FUNCTION_BLOCK VariableToEvent (* Basic Function Block Type *)
  (* Standard: 61499-2 *)
  (* Version 0.2, 2003-12-04, JHC, Rockwell Automation, Renamed for better indexing. *)
  (* Version 0.1, 2002-11-05, JHC, Rockwell Automation, Corrected missing ST element in Algorithm REQ. *)
  (* Version 0.0, 2000-05-30, JHC, Rockwell Automation *)
  (* Compiler header: package fb.rt.cs725; *)
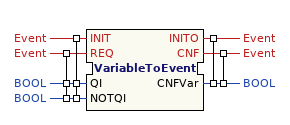
  EVENT_INPUT
    INIT WITH QI, NOTQI; (* Initialization Request *)
    REQ WITH QI, NOTQI; (* Normal Execution Request *)
  END_EVENT
  EVENT_OUTPUT
    INITO WITH CNFVar; (* Initialization Confirm *)
    CNF WITH CNFVar; (* Execution Confirmation *)
  END_EVENT
  VAR_INPUT
    QI : BOOL; (* Input event qualifier *)
    NOTQI : BOOL;
  END_VAR
  VAR_OUTPUT
    CNFVar : BOOL;
  END_VAR
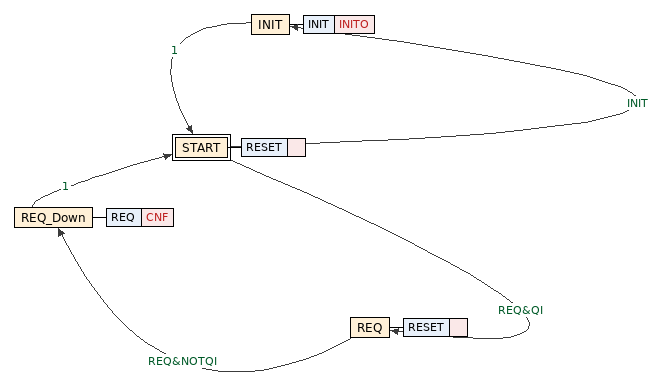
  EC_STATES
    START : RESET; (* Initial State *)
    INIT : INIT -> INITO; (* Initialization *)
    REQ : RESET; (* Normal execution *)
    REQ_Down : REQ -> CNF;
  END_STATES
  EC_TRANSITIONS
    START TO INIT := INIT;
    INIT TO START := 1;
    START TO REQ := REQ&QI;
    REQ TO REQ_Down := REQ&NOTQI;
    REQ_Down TO START := 1;
  END_TRANSITIONS
  ALGORITHM INIT IN Java: (* Initialization algorithm *)
CNFVar.value = false;
  END_ALGORITHM
  ALGORITHM REQ IN Java: (* Normally executed algorithm *)
CNFVar.value = true;
System.out.println(this + "PE CHANGED!!!");
  END_ALGORITHM
  ALGORITHM RESET IN Java:
CNFVar.value=false;
System.out.println(this+"PE RESET/NOT CHANGED!!!");
  END_ALGORITHM
END_FUNCTION_BLOCK
